// TIA Portal V17 export
// export: Created 2022-07-20T07:01:27.7836548Z, ExportSetting WithDefaults, DisplayName Totally Integrated Automation Portal, DisplayVersion V17, DisplayName TIA Portal Openness, DisplayVersion V17, DisplayName TIA Portal Version Control Interface, DisplayVersion V17, DisplayName SINAMICS Startdrive Advanced, DisplayVersion V17, DisplayName SINAMICS Startdrive G130, G150, S120, S150, SINAMICS MV, S210, DisplayVersion V17, DisplayName SINAMICS Startdrive G110M, G120, G120C, G120D, G120P, G115D, DisplayVersion V17, DisplayName STEP 7 Professional, DisplayVersion V17, DisplayName STEP 7 Safety, DisplayVersion V17, DisplayName WinCC Advanced, DisplayVersion V17
FUNCTION_BLOCK "FB10181_ChucksFSManager"   // FB10181, LAD
{ S7_Optimized_Access := 'TRUE' }
VERSION : 0.1
// stored: AutoNumber false, IsIECCheckEnabled false, IsRetainMemResEnabled false, MemoryReserve 100, SetENOAutomatically false, UDAEnableTagReadback false
   VAR_INPUT
      WorkingMode : Bool;
      BypassMode : Bool;
      Input_ChuckInPosition : Bool;
      Input_AuthorisationToStart : Bool;
      AuthorisationToStartTime : Time;
   END_VAR
   VAR_OUTPUT
      Output_ChucksInPosition : Bool;
      Output_AuthorisationToStart : Bool;
   END_VAR
   VAR
      TON_AuthorisationToStartTimer : TON_TIME;
      TON_SafetyChucksToStart { S7_SetPoint := 'True'} : TON_TIME;
   END_VAR
BEGIN

REGION Network 1 (SCL): First Scan
   IF "FirstScan" THEN
       ;
   END_IF;
END_REGION

REGION Network 2 (SCL): Edge Signals & Timers
   REGION EDGE SIGNALS

   END_REGION

   REGION TIMERS
       #TON_AuthorisationToStartTimer(IN := NOT(#Input_ChuckInPosition),
                                      PT := #AuthorisationToStartTime);
       #TON_SafetyChucksToStart(IN := #WorkingMode AND NOT (#Input_ChuckInPosition),
                                PT := T#400ms); //Pas besoin
   END_REGION
END_REGION

REGION Network 3 (SCL): Chucks FS Management
   IF #BypassMode THEN
       #Output_ChucksInPosition := TRUE;
       #Output_AuthorisationToStart := #TON_AuthorisationToStartTimer.Q;
   ELSIF #WorkingMode THEN
       #Output_ChucksInPosition := #Input_ChuckInPosition;
       #Output_AuthorisationToStart := #Input_AuthorisationToStart;
   END_IF;
END_REGION
END_FUNCTION_BLOCK
